# EPICS autosave request: LabJackApp/Db/LabJack_device_settings.req
$(P)PollSleepMS
$(P)AiAllSettlingUS
